FUNCTION_BLOCK FB_LimSwStatus IMPLEMENTS I_LimSwStatus
VAR_INPUT
END_VAR
VAR_OUTPUT
END_VAR
VAR
    (* Hardware *)
   // NC Forward Limit Switch: TRUE if ok to move
    bLimitForwardEnable AT %I*: BOOL;
    // NC Backward Limit Switch: TRUE if ok to move
    bLimitBackwardEnable AT %I*: BOOL;
    // NO Home Switch: TRUE if at home
    bLimitHome AT %I*: BOOL;

END_VAR

PROPERTY LimBackward : BOOL
GET
LimBackward := bLimitBackwardEnable;
END_GET
SET
bLimitBackwardEnable :=LimBackward;
END_SET
END_PROPERTY

PROPERTY LimForward : BOOL
GET
LimForward := bLimitForwardEnable;
END_GET
SET
bLimitForwardEnable := LimForward;
END_SET
END_PROPERTY

PROPERTY LimHome : BOOL
GET
LimHome :=  bLimitHome ;
END_GET
END_PROPERTY

END_FUNCTION_BLOCK

(* stored: Version 1.1.0.1
   POU FB_LimSwStatus: Id {322e8186-deb9-4a53-b303-d1d3662306db}, SpecialFunc None
   Property LimBackward: Id {35aa245a-d874-4916-85c5-42c60fad40f0}
   Get Get: Id {5fbf77a3-1565-4123-a7e4-8abd4560ecb2}
   Set Set: Id {bd1cd8be-0ef5-4bb3-be52-2ca7a979245c}
   Property LimForward: Id {60bb8d48-4b37-425b-923e-b1e7d0d2cba8}
   Get Get: Id {c6fce77e-af19-46cd-b898-ad9a07ade412}
   Set Set: Id {7860d5f2-6502-460a-9e8f-7946aad41f2e}
   Property LimHome: Id {1b597d59-cd48-4a23-82a2-a38399b4eb9e}
   Get Get: Id {a5e85be1-90e3-408d-830c-f40a8296404c} *)
